TYPE T_HashTableEntry :
STRUCT
    {attribute 'pytmc' := '
        pv: Key
        io: i
     '}
    key : DWORD := 0;
    value : PVOID := 0;
END_STRUCT
END_TYPE

(* stored: Version 1.1.0.1
   DUT T_HashTableEntry: Id {981738f9-cdaa-4fe1-95f5-e01133a08af9} *)
